{attribute 'qualified_only'}
{attribute 'strict'}
{attribute 'to_string'}
TYPE E_RESET_ORIGIN :
(
	UNDEFINED := 0,
	
	CONTROL_AREA_MANUAL,	// Operator presses reset on the control signal
	
	CONTROL_AREA_AUTO,		// Automatic (external) reset, eg. doors were closed and a reset was triggered

	EXTERNAL,				// Through FB input, eg. hard wired button or banner reset
	
	ALARM_SPECIFIC			// Specific device/alarm reset 
);
END_TYPE

(* stored: Version 1.1.0.1, ProductVersion 3.1.4026.18
   DUT E_RESET_ORIGIN: Id {7580b49d-68bd-4586-ad6f-a0e71e28c011} *)
